(* Logix 5000 project; controller AdvManLab vendor 1 type 14 code 158 rev 28.12; software revision 28.01; part 10 of 13 *)
(* tags used below, declared in another part *)
   R6Z_Assign : BOOL;
   R6Z_Check_InProgress : BOOL;
   R6Z_Check_Part_NO : SINT;
   R6Z_Check_Read : BOOL;
   R6Z_Check_Results : BOOL;
   R6Z_Check_Start : BOOL;
   R6Z_Clear_All : BOOL;
   R6Z_Clear_All_Inprogress : BOOL;
   R6Z_Clear_All_Start : BOOL;
   R6Z_Current_Part_NO : SINT;
   R6Z_Current_Process_NO : SINT;
   R6Z_Part_Type_Counter : SINT;
   R6Z_Process : BOOL;
   R6Z_Read : BOOL;
   R6Z_Read_Check_Fail : BOOL;
   R6Z_Read_Check_InProgress : BOOL;
   R6Z_Read_Check_Results : BOOL;
   R6Z_Read_Check_Start : BOOL;
   R6Z_Read_Finished : BOOL;
   R6Z_Read_InProgress : BOOL;
   R6Z_Read_Results : BOOL;
   R6Z_Read_Start : BOOL;
   R6Z_Write : BOOL;
   R6Z_Write_Finished_Check : BOOL;
   R6Z_Write_Inprogress : BOOL;
   R6Z_Write_Pass : BOOL;
   Cell_2 : Fanuc_Cell;
   CNC_3_Done : BOOL;   // CNC 3 has completed cutting the part
   CNC_4_Done : BOOL;   // CNC 4 has completed cutting the part
   Enable_Process_Update : BOOL;
   Mode_Auto : BOOL;
   Mode_Semi : BOOL;
   Mode_Start : BOOL;
   R2Z_Current_Part_NO : DINT;
   R2Z_Current_Process_NO : DINT;
   R2Z_Read : BOOL;
   R2Z_Read_Finished : BOOL;
   R2Z_Read_InProgress : BOOL;
   R2Z_Read_Results : BOOL;
   R2Z_Read_Start : BOOL;
   R3J_Assign : BOOL;
   R3J_Check_Process_NO : DINT;
   R3J_Current_Part_NO : SINT;
   R3J_Current_Process_NO : SINT;
   R3J_Process : BOOL;
   R3J_Read : BOOL;
   R3J_Read_Check_Fail : BOOL;
   R3J_Read_Check_InProgress : BOOL;
   R3J_Read_Check_Results : BOOL;
   R3J_Read_Check_Start : BOOL;
   R3J_Read_Finished : BOOL;
   R3J_Read_InProgress : BOOL;
   R3J_Read_Results : BOOL;
   R3J_Read_Start : BOOL;
   R3J_Write : BOOL;
   R3J_Write_Finished_Check : BOOL;
   R3J_Write_Inprogress : BOOL;
   R3J_Write_Pass : BOOL;
   R5Z_Current_Part_NO : DINT;
   R5Z_Current_Process_NO : DINT;
   R5Z_Read : BOOL;
   R5Z_Read_Finished : BOOL;
   R5Z_Read_InProgress : BOOL;
   R5Z_Read_Results : BOOL;
   R5Z_Read_Start : BOOL;
   R6S_Check_Current_Part_NO : DINT;
   R6S_Check_Current_Process_NO : DINT;
   R6S_User_Input_Part_NO : DINT;
   R6S_User_Input_Process_NO : DINT;
   R6Z_Check_Read_PB : BOOL;
   R6Z_Clear_All_PB : BOOL;
   R6Z_Write_Check : BOOL;
   R6Z_Write_Check_1 : BOOL;
   R6Z_Write_Inprogress_Check : BOOL;
   R6Z_Write_Inprogress_Check_1 : BOOL;
   R6Z_Write_Test : BOOL;
   R6Z_Write_Test_1 : BOOL;
   R6Z_Write_Test_PB : BOOL;
   RFIDTP2 : ALIAS FOR RFID_N054:I.Channel[1].TagPresent;   // RFID Tag at Cell 2 Hold Back Stop
   RFIDTP3 : ALIAS FOR RFID_N055:I.Channel[0].TagPresent;   // RFID Tag at Cell 2 Stop
   RFIDTP5 : ALIAS FOR RFID_N056:I.Channel[0].TagPresent;   // RFID Tag at Cell 3 Stop
   RFIDTP6 : ALIAS FOR RFID_N056:I.Channel[1].TagPresent;
   Robot2_DroppedP3 : BOOL;
   Robot2_DroppedP4 : BOOL;
   Robot2DroppedPart : BOOL;
(* MainProgram, continued *)

ROUTINE RFID_2_ZZ   (* ladder *)
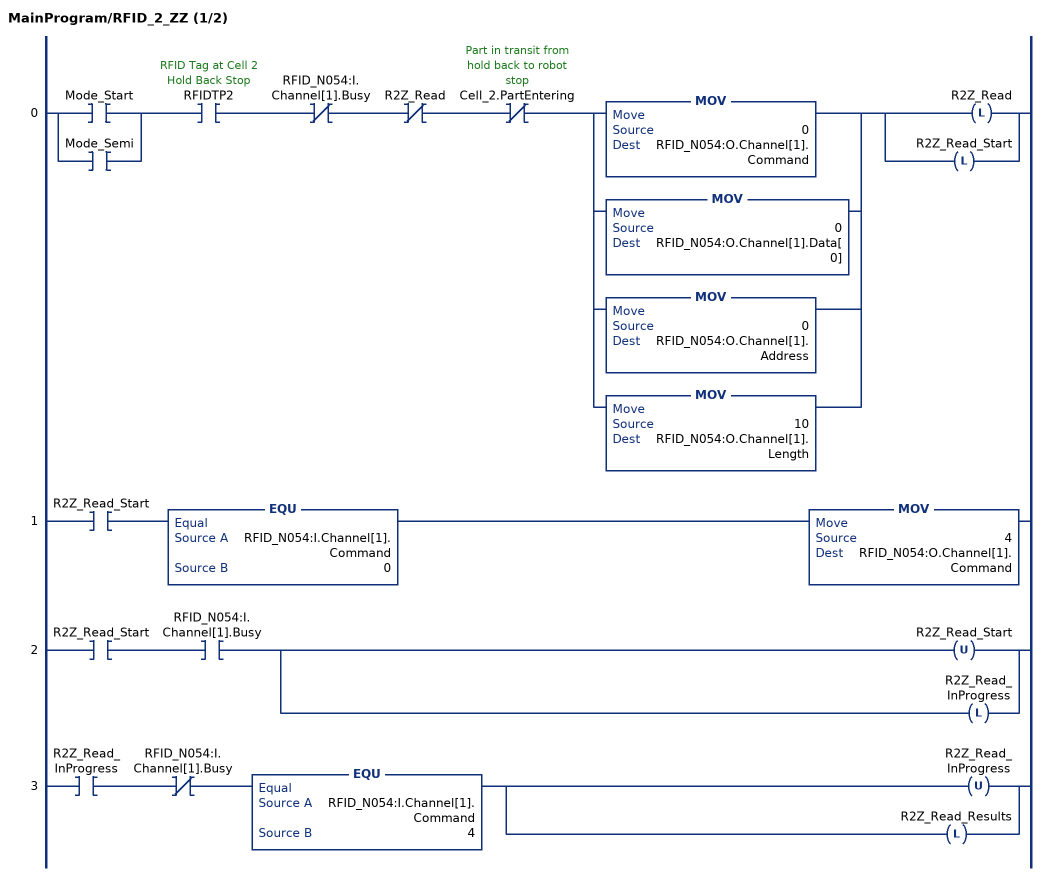
   0: [XIC(Mode_Start) ,XIC(Mode_Semi) ]XIC(RFIDTP2)XIO(RFID_N054:I.Channel[1].Busy)XIO(R2Z_Read)XIO(Cell_2.PartEntering)[MOV(0,RFID_N054:O.Channel[1].Command) ,MOV(0,RFID_N054:O.Channel[1].Data[0]) ,MOV(0,RFID_N054:O.Channel[1].Address) ,MOV(10,RFID_N054:O.Channel[1].Length) ][OTL(R2Z_Read) ,OTL(R2Z_Read_Start) ];
   1: XIC(R2Z_Read_Start)EQU(RFID_N054:I.Channel[1].Command,0)MOV(4,RFID_N054:O.Channel[1].Command);
   2: XIC(R2Z_Read_Start)XIC(RFID_N054:I.Channel[1].Busy)[OTU(R2Z_Read_Start) ,OTL(R2Z_Read_InProgress) ];
   3: XIC(R2Z_Read_InProgress)XIO(RFID_N054:I.Channel[1].Busy)EQU(RFID_N054:I.Channel[1].Command,4)[OTU(R2Z_Read_InProgress) ,OTL(R2Z_Read_Results) ];
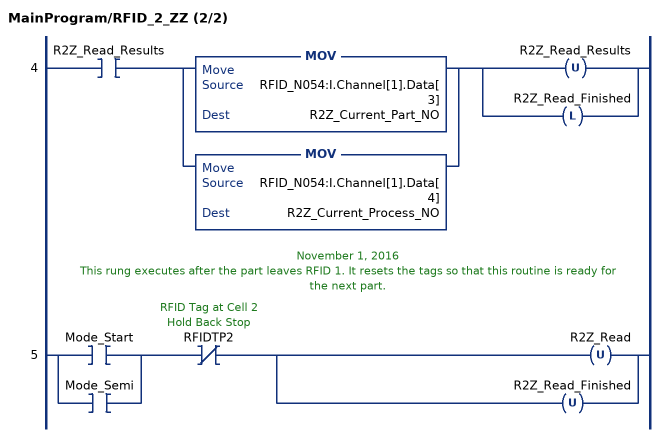
   4: XIC(R2Z_Read_Results)[MOV(RFID_N054:I.Channel[1].Data[3],R2Z_Current_Part_NO) ,MOV(RFID_N054:I.Channel[1].Data[4],R2Z_Current_Process_NO) ][OTU(R2Z_Read_Results) ,OTL(R2Z_Read_Finished) ];
   // November 1, 2016
   // This rung executes after the part leaves RFID 1. It resets the tags so that this routine is ready for the next part.
   5: [XIC(Mode_Start) ,XIC(Mode_Semi) ]XIO(RFIDTP2)[OTU(R2Z_Read) ,OTU(R2Z_Read_Finished) ];
END_ROUTINE

ROUTINE RFID_3_JW   (* ladder *)
// Rewrite of RFID_3 using new read/write logic of RFID_6_ZZ
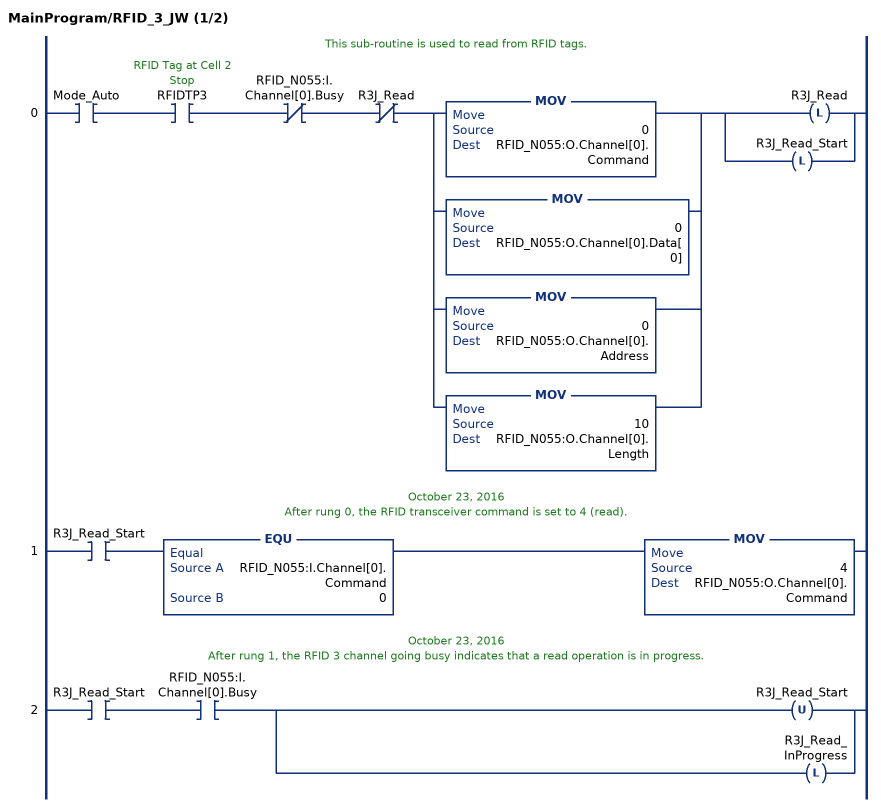
   // This sub-routine is used to read from RFID tags.
   0: XIC(Mode_Auto)XIC(RFIDTP3)XIO(RFID_N055:I.Channel[0].Busy)XIO(R3J_Read)[MOV(0,RFID_N055:O.Channel[0].Command) ,MOV(0,RFID_N055:O.Channel[0].Data[0]) ,MOV(0,RFID_N055:O.Channel[0].Address) ,MOV(10,RFID_N055:O.Channel[0].Length) ][OTL(R3J_Read) ,OTL(R3J_Read_Start) ];
   // October 23, 2016
   // After rung 0, the RFID transceiver command is set to 4 (read).
   1: XIC(R3J_Read_Start)EQU(RFID_N055:I.Channel[0].Command,0)MOV(4,RFID_N055:O.Channel[0].Command);
   // October 23, 2016
   // After rung 1, the RFID 3 channel going busy indicates that a read operation is in progress.
   2: XIC(R3J_Read_Start)XIC(RFID_N055:I.Channel[0].Busy)[OTU(R3J_Read_Start) ,OTL(R3J_Read_InProgress) ];
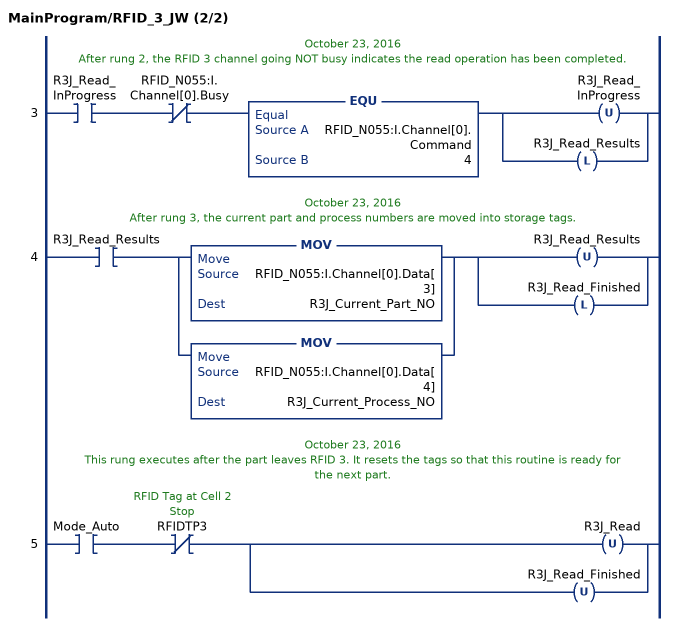
   // October 23, 2016
   // After rung 2, the RFID 3 channel going NOT busy indicates the read operation has been completed.
   3: XIC(R3J_Read_InProgress)XIO(RFID_N055:I.Channel[0].Busy)EQU(RFID_N055:I.Channel[0].Command,4)[OTU(R3J_Read_InProgress) ,OTL(R3J_Read_Results) ];
   // October 23, 2016
   // After rung 3, the current part and process numbers are moved into storage tags.
   4: XIC(R3J_Read_Results)[MOV(RFID_N055:I.Channel[0].Data[3],R3J_Current_Part_NO) ,MOV(RFID_N055:I.Channel[0].Data[4],R3J_Current_Process_NO) ][OTU(R3J_Read_Results) ,OTL(R3J_Read_Finished) ];
   // October 23, 2016
   // This rung executes after the part leaves RFID 3. It resets the tags so that this routine is ready for the next part.
   5: XIC(Mode_Auto)XIO(RFIDTP3)[OTU(R3J_Read) ,OTU(R3J_Read_Finished) ];
END_ROUTINE

ROUTINE RFID_5_ZZ   (* ladder *)
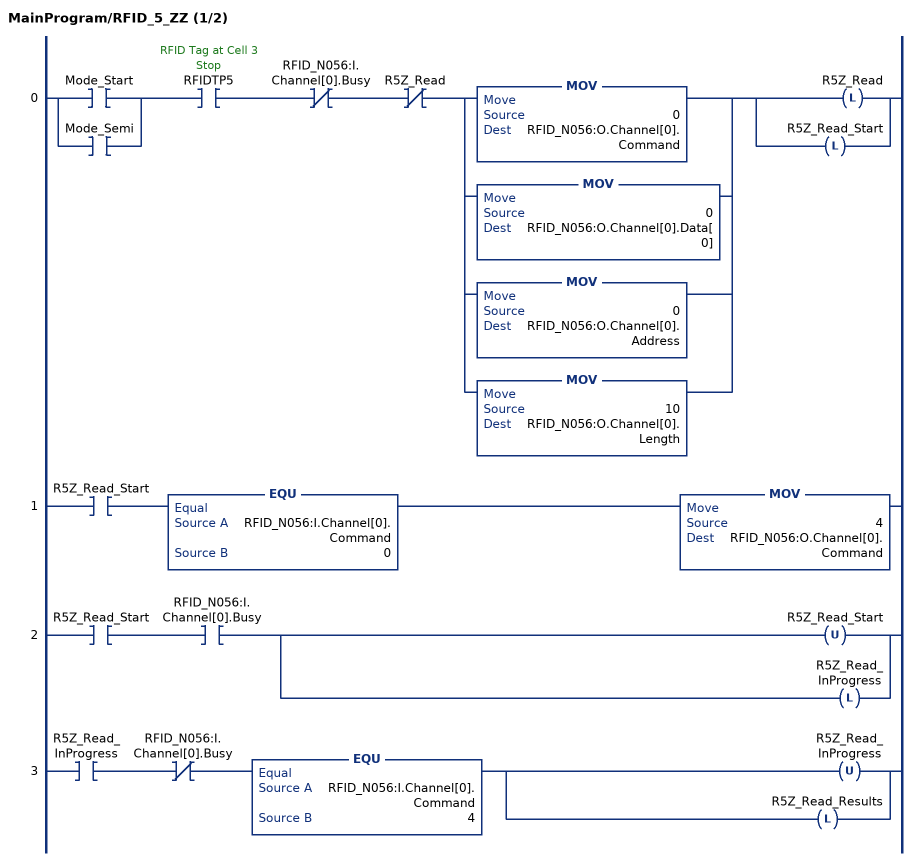
   0: [XIC(Mode_Start) ,XIC(Mode_Semi) ]XIC(RFIDTP5)XIO(RFID_N056:I.Channel[0].Busy)XIO(R5Z_Read)[MOV(0,RFID_N056:O.Channel[0].Command) ,MOV(0,RFID_N056:O.Channel[0].Data[0]) ,MOV(0,RFID_N056:O.Channel[0].Address) ,MOV(10,RFID_N056:O.Channel[0].Length) ][OTL(R5Z_Read) ,OTL(R5Z_Read_Start) ];
   1: XIC(R5Z_Read_Start)EQU(RFID_N056:I.Channel[0].Command,0)MOV(4,RFID_N056:O.Channel[0].Command);
   2: XIC(R5Z_Read_Start)XIC(RFID_N056:I.Channel[0].Busy)[OTU(R5Z_Read_Start) ,OTL(R5Z_Read_InProgress) ];
   3: XIC(R5Z_Read_InProgress)XIO(RFID_N056:I.Channel[0].Busy)EQU(RFID_N056:I.Channel[0].Command,4)[OTU(R5Z_Read_InProgress) ,OTL(R5Z_Read_Results) ];
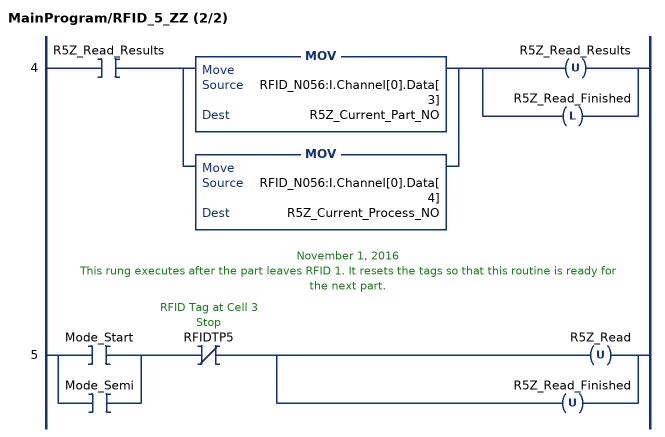
   4: XIC(R5Z_Read_Results)[MOV(RFID_N056:I.Channel[0].Data[3],R5Z_Current_Part_NO) ,MOV(RFID_N056:I.Channel[0].Data[4],R5Z_Current_Process_NO) ][OTU(R5Z_Read_Results) ,OTL(R5Z_Read_Finished) ];
   // November 1, 2016
   // This rung executes after the part leaves RFID 1. It resets the tags so that this routine is ready for the next part.
   5: [XIC(Mode_Start) ,XIC(Mode_Semi) ]XIO(RFIDTP5)[OTU(R5Z_Read) ,OTU(R5Z_Read_Finished) ];
END_ROUTINE

ROUTINE RFID_6_Clear_All_ZZ   (* ladder *)
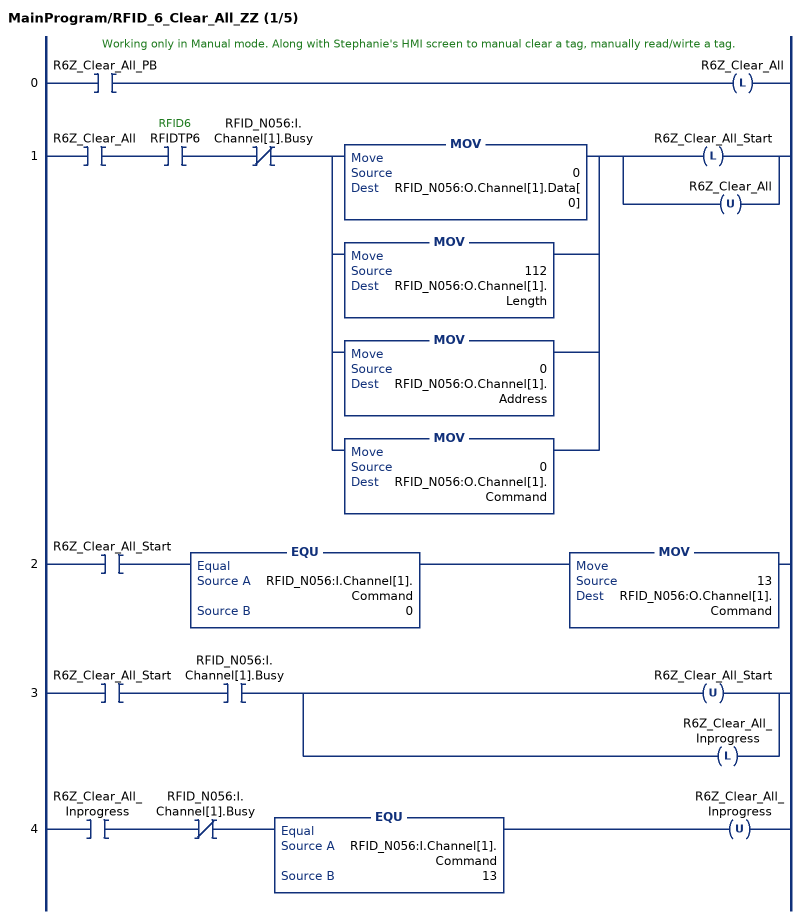
   // Working only in Manual mode. Along with Stephanie's HMI screen to manual clear a tag, manually read/wirte a tag.
   0: XIC(R6Z_Clear_All_PB)OTL(R6Z_Clear_All);
   1: XIC(R6Z_Clear_All)XIC(RFIDTP6)XIO(RFID_N056:I.Channel[1].Busy)[MOV(0,RFID_N056:O.Channel[1].Data[0]) ,MOV(112,RFID_N056:O.Channel[1].Length) ,MOV(0,RFID_N056:O.Channel[1].Address) ,MOV(0,RFID_N056:O.Channel[1].Command) ][OTL(R6Z_Clear_All_Start) ,OTU(R6Z_Clear_All) ];
   2: XIC(R6Z_Clear_All_Start)EQU(RFID_N056:I.Channel[1].Command,0)MOV(13,RFID_N056:O.Channel[1].Command);
   3: XIC(R6Z_Clear_All_Start)XIC(RFID_N056:I.Channel[1].Busy)[OTU(R6Z_Clear_All_Start) ,OTL(R6Z_Clear_All_Inprogress) ];
   4: XIC(R6Z_Clear_All_Inprogress)XIO(RFID_N056:I.Channel[1].Busy)EQU(RFID_N056:I.Channel[1].Command,13)OTU(R6Z_Clear_All_Inprogress);
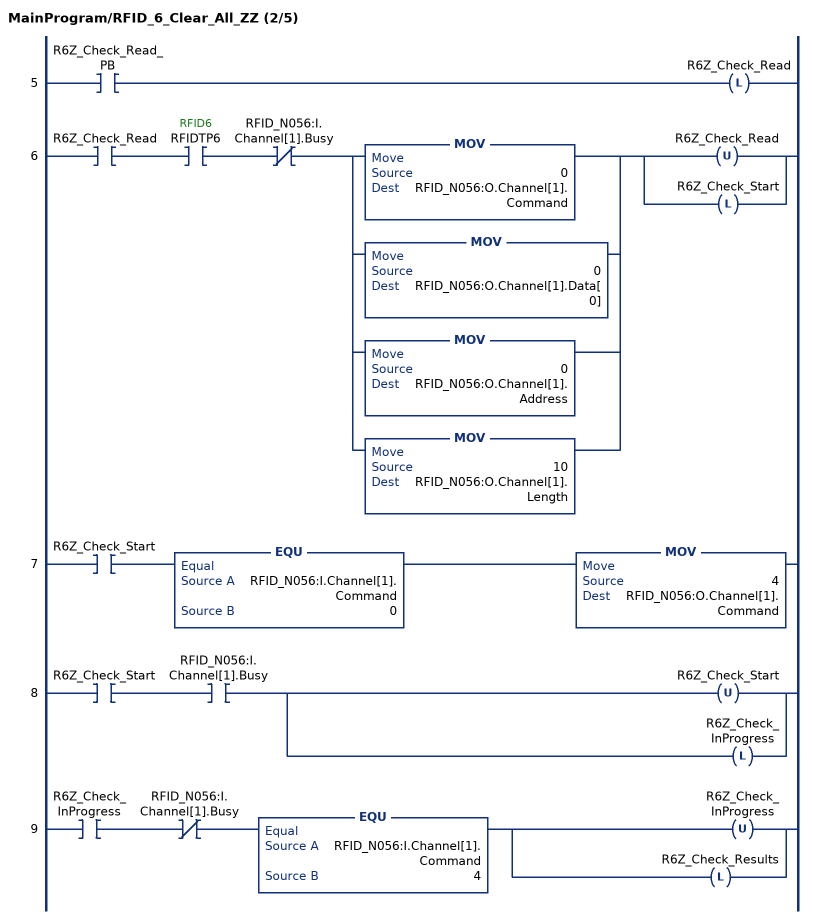
   5: XIC(R6Z_Check_Read_PB)OTL(R6Z_Check_Read);
   6: XIC(R6Z_Check_Read)XIC(RFIDTP6)XIO(RFID_N056:I.Channel[1].Busy)[MOV(0,RFID_N056:O.Channel[1].Command) ,MOV(0,RFID_N056:O.Channel[1].Data[0]) ,MOV(0,RFID_N056:O.Channel[1].Address) ,MOV(10,RFID_N056:O.Channel[1].Length) ][OTU(R6Z_Check_Read) ,OTL(R6Z_Check_Start) ];
   7: XIC(R6Z_Check_Start)EQU(RFID_N056:I.Channel[1].Command,0)MOV(4,RFID_N056:O.Channel[1].Command);
   8: XIC(R6Z_Check_Start)XIC(RFID_N056:I.Channel[1].Busy)[OTU(R6Z_Check_Start) ,OTL(R6Z_Check_InProgress) ];
   9: XIC(R6Z_Check_InProgress)XIO(RFID_N056:I.Channel[1].Busy)EQU(RFID_N056:I.Channel[1].Command,4)[OTU(R6Z_Check_InProgress) ,OTL(R6Z_Check_Results) ];
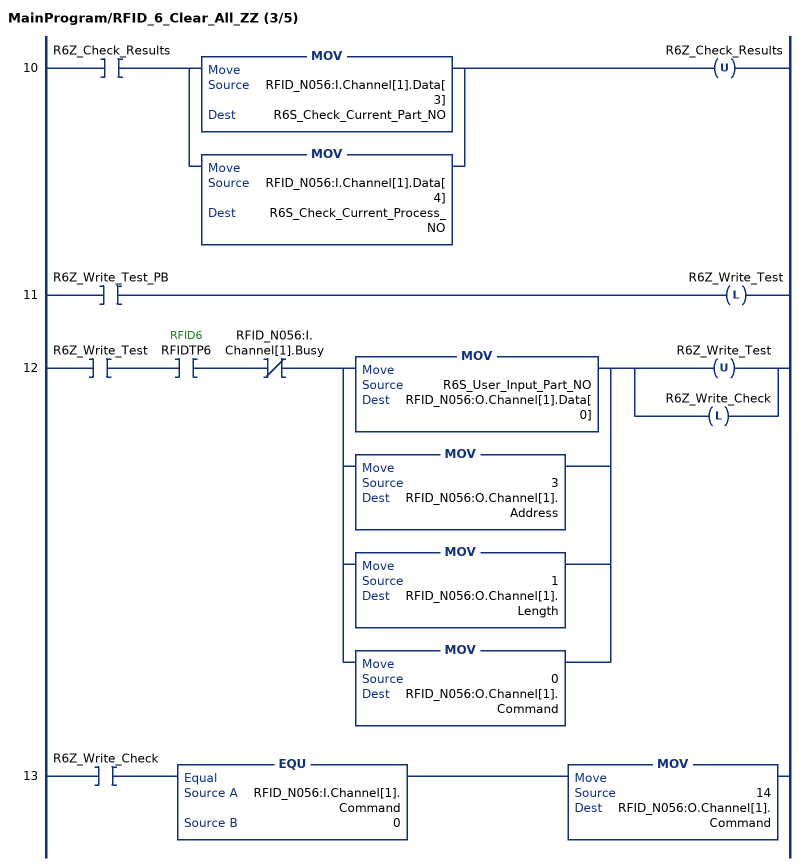
   10: XIC(R6Z_Check_Results)[MOV(RFID_N056:I.Channel[1].Data[3],R6S_Check_Current_Part_NO) ,MOV(RFID_N056:I.Channel[1].Data[4],R6S_Check_Current_Process_NO) ]OTU(R6Z_Check_Results);
   11: XIC(R6Z_Write_Test_PB)OTL(R6Z_Write_Test);
   12: XIC(R6Z_Write_Test)XIC(RFIDTP6)XIO(RFID_N056:I.Channel[1].Busy)[MOV(R6S_User_Input_Part_NO,RFID_N056:O.Channel[1].Data[0]) ,MOV(3,RFID_N056:O.Channel[1].Address) ,MOV(1,RFID_N056:O.Channel[1].Length) ,MOV(0,RFID_N056:O.Channel[1].Command) ][OTU(R6Z_Write_Test) ,OTL(R6Z_Write_Check) ];
   13: XIC(R6Z_Write_Check)EQU(RFID_N056:I.Channel[1].Command,0)MOV(14,RFID_N056:O.Channel[1].Command);
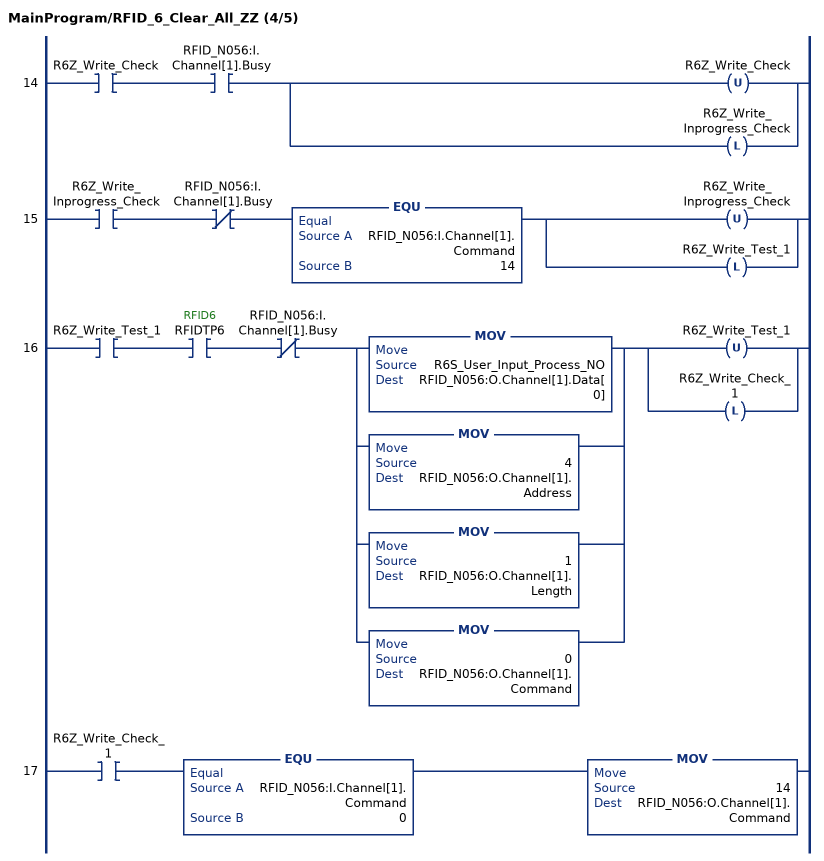
   14: XIC(R6Z_Write_Check)XIC(RFID_N056:I.Channel[1].Busy)[OTU(R6Z_Write_Check) ,OTL(R6Z_Write_Inprogress_Check) ];
   15: XIC(R6Z_Write_Inprogress_Check)XIO(RFID_N056:I.Channel[1].Busy)EQU(RFID_N056:I.Channel[1].Command,14)[OTU(R6Z_Write_Inprogress_Check) ,OTL(R6Z_Write_Test_1) ];
   16: XIC(R6Z_Write_Test_1)XIC(RFIDTP6)XIO(RFID_N056:I.Channel[1].Busy)[MOV(R6S_User_Input_Process_NO,RFID_N056:O.Channel[1].Data[0]) ,MOV(4,RFID_N056:O.Channel[1].Address) ,MOV(1,RFID_N056:O.Channel[1].Length) ,MOV(0,RFID_N056:O.Channel[1].Command) ][OTU(R6Z_Write_Test_1) ,OTL(R6Z_Write_Check_1) ];
   17: XIC(R6Z_Write_Check_1)EQU(RFID_N056:I.Channel[1].Command,0)MOV(14,RFID_N056:O.Channel[1].Command);
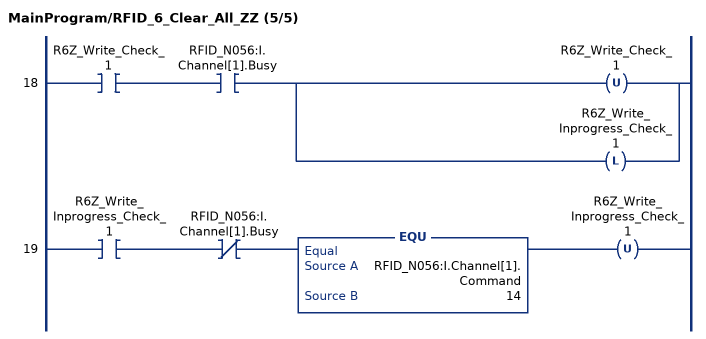
   18: XIC(R6Z_Write_Check_1)XIC(RFID_N056:I.Channel[1].Busy)[OTU(R6Z_Write_Check_1) ,OTL(R6Z_Write_Inprogress_Check_1) ];
   19: XIC(R6Z_Write_Inprogress_Check_1)XIO(RFID_N056:I.Channel[1].Busy)EQU(RFID_N056:I.Channel[1].Command,14)OTU(R6Z_Write_Inprogress_Check_1);
END_ROUTINE

ROUTINE RFID_6_ZZ   (* ladder *)
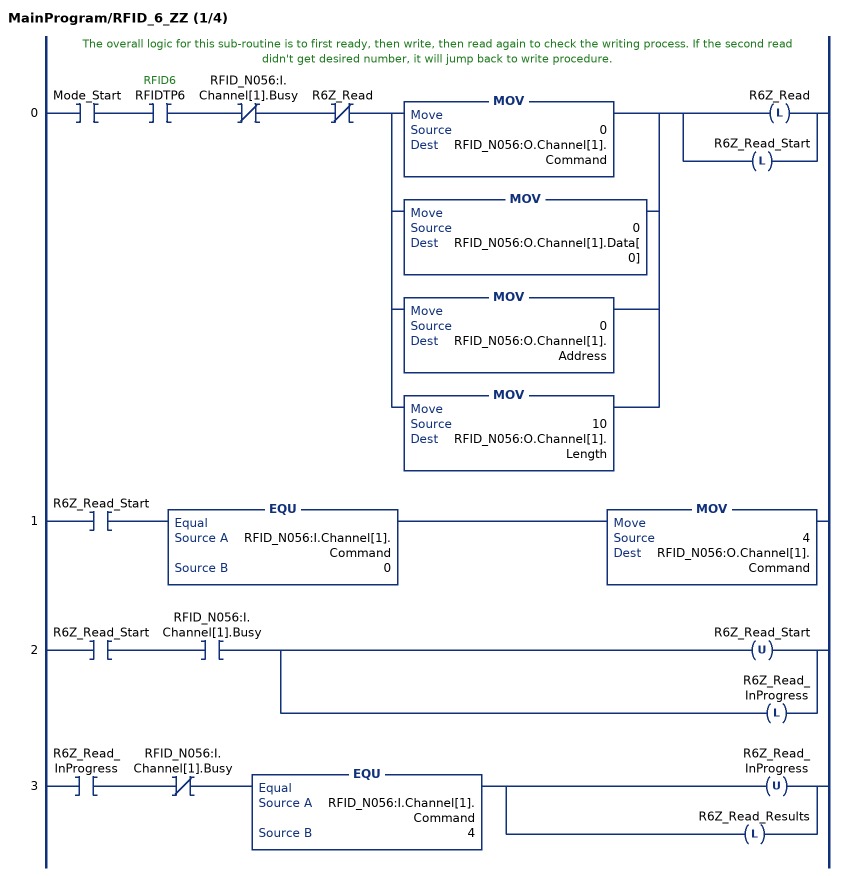
   // The overall logic for this sub-routine is to first ready, then write, then read again to check the writing process. If the second read didn't get desired number, it will jump back to write procedure.
   0: XIC(Mode_Start)XIC(RFIDTP6)XIO(RFID_N056:I.Channel[1].Busy)XIO(R6Z_Read)[MOV(0,RFID_N056:O.Channel[1].Command) ,MOV(0,RFID_N056:O.Channel[1].Data[0]) ,MOV(0,RFID_N056:O.Channel[1].Address) ,MOV(10,RFID_N056:O.Channel[1].Length) ][OTL(R6Z_Read) ,OTL(R6Z_Read_Start) ];
   1: XIC(R6Z_Read_Start)EQU(RFID_N056:I.Channel[1].Command,0)MOV(4,RFID_N056:O.Channel[1].Command);
   2: XIC(R6Z_Read_Start)XIC(RFID_N056:I.Channel[1].Busy)[OTU(R6Z_Read_Start) ,OTL(R6Z_Read_InProgress) ];
   3: XIC(R6Z_Read_InProgress)XIO(RFID_N056:I.Channel[1].Busy)EQU(RFID_N056:I.Channel[1].Command,4)[OTU(R6Z_Read_InProgress) ,OTL(R6Z_Read_Results) ];
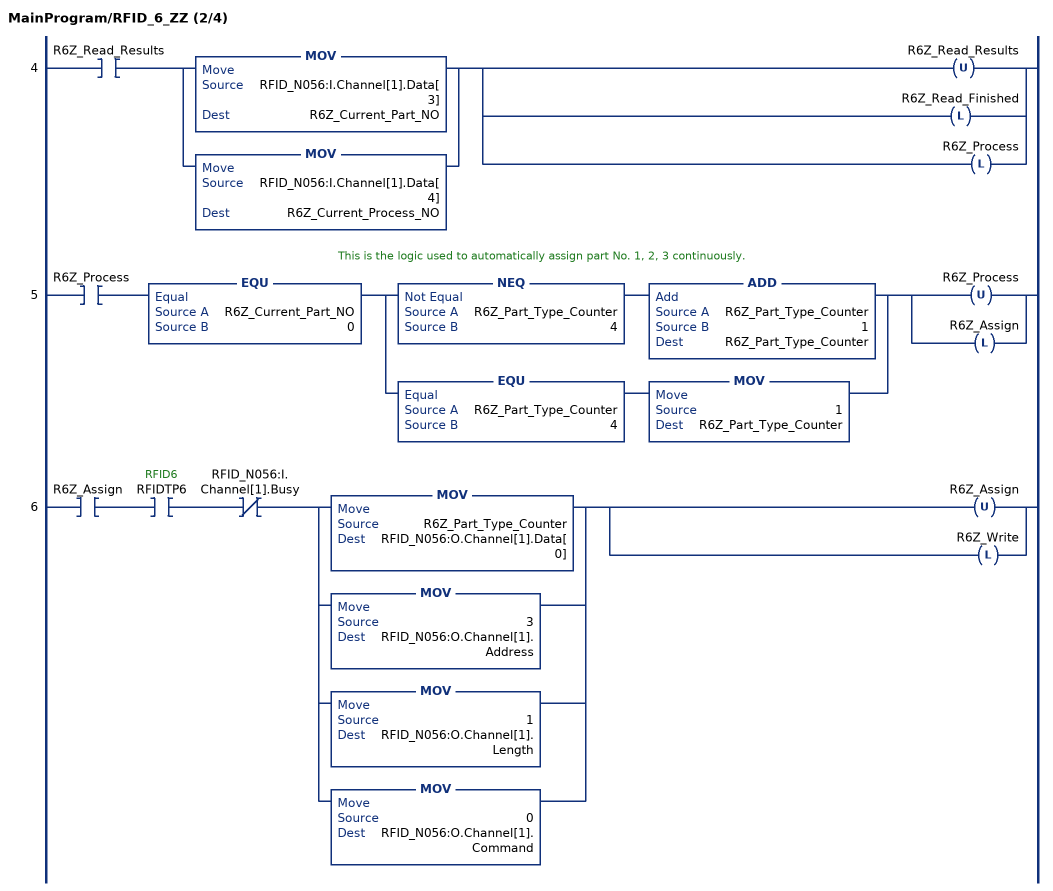
   4: XIC(R6Z_Read_Results)[MOV(RFID_N056:I.Channel[1].Data[3],R6Z_Current_Part_NO) ,MOV(RFID_N056:I.Channel[1].Data[4],R6Z_Current_Process_NO) ][OTU(R6Z_Read_Results) ,OTL(R6Z_Read_Finished) ,OTL(R6Z_Process) ];
   // This is the logic used to automatically assign part No. 1, 2, 3 continuously.
   5: XIC(R6Z_Process)EQU(R6Z_Current_Part_NO,0)[NEQ(R6Z_Part_Type_Counter,4) ADD(R6Z_Part_Type_Counter,1,R6Z_Part_Type_Counter) ,EQU(R6Z_Part_Type_Counter,4) MOV(1,R6Z_Part_Type_Counter) ][OTU(R6Z_Process) ,OTL(R6Z_Assign) ];
   6: XIC(R6Z_Assign)XIC(RFIDTP6)XIO(RFID_N056:I.Channel[1].Busy)[MOV(R6Z_Part_Type_Counter,RFID_N056:O.Channel[1].Data[0]) ,MOV(3,RFID_N056:O.Channel[1].Address) ,MOV(1,RFID_N056:O.Channel[1].Length) ,MOV(0,RFID_N056:O.Channel[1].Command) ][OTU(R6Z_Assign) ,OTL(R6Z_Write) ];
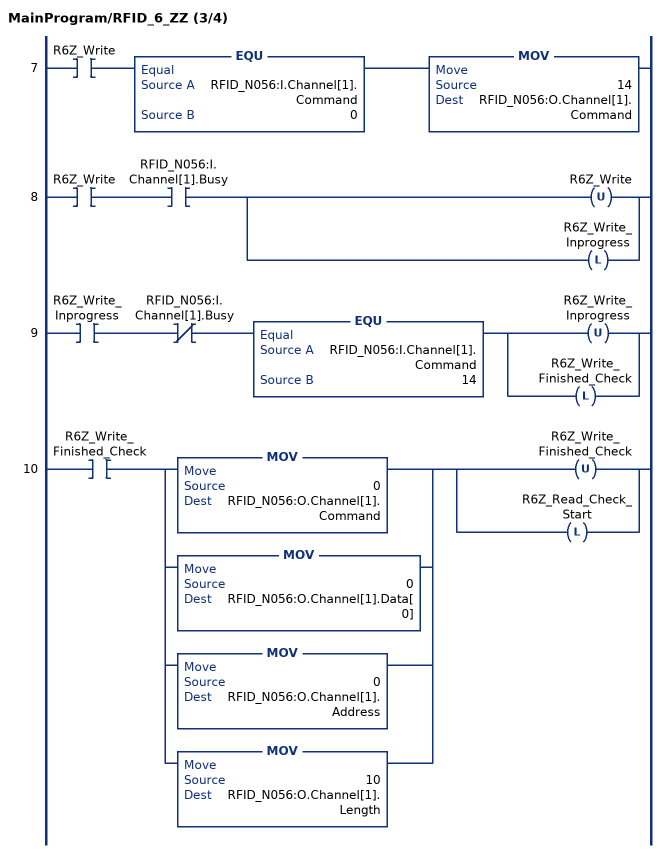
   7: XIC(R6Z_Write)EQU(RFID_N056:I.Channel[1].Command,0)MOV(14,RFID_N056:O.Channel[1].Command);
   8: XIC(R6Z_Write)XIC(RFID_N056:I.Channel[1].Busy)[OTU(R6Z_Write) ,OTL(R6Z_Write_Inprogress) ];
   9: XIC(R6Z_Write_Inprogress)XIO(RFID_N056:I.Channel[1].Busy)EQU(RFID_N056:I.Channel[1].Command,14)[OTU(R6Z_Write_Inprogress) ,OTL(R6Z_Write_Finished_Check) ];
   10: XIC(R6Z_Write_Finished_Check)[MOV(0,RFID_N056:O.Channel[1].Command) ,MOV(0,RFID_N056:O.Channel[1].Data[0]) ,MOV(0,RFID_N056:O.Channel[1].Address) ,MOV(10,RFID_N056:O.Channel[1].Length) ][OTU(R6Z_Write_Finished_Check) ,OTL(R6Z_Read_Check_Start) ];
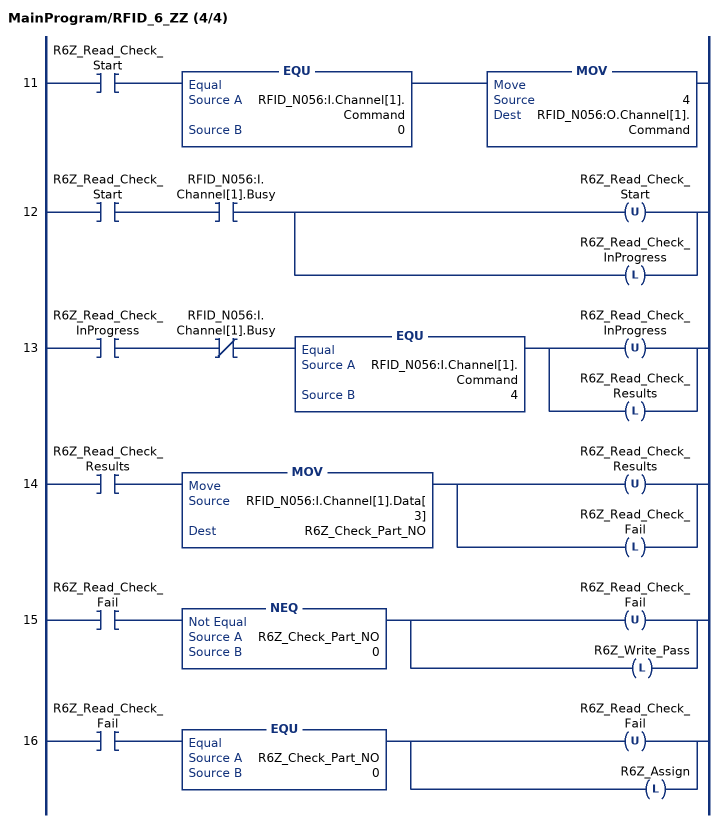
   11: XIC(R6Z_Read_Check_Start)EQU(RFID_N056:I.Channel[1].Command,0)MOV(4,RFID_N056:O.Channel[1].Command);
   12: XIC(R6Z_Read_Check_Start)XIC(RFID_N056:I.Channel[1].Busy)[OTU(R6Z_Read_Check_Start) ,OTL(R6Z_Read_Check_InProgress) ];
   13: XIC(R6Z_Read_Check_InProgress)XIO(RFID_N056:I.Channel[1].Busy)EQU(RFID_N056:I.Channel[1].Command,4)[OTU(R6Z_Read_Check_InProgress) ,OTL(R6Z_Read_Check_Results) ];
   14: XIC(R6Z_Read_Check_Results)MOV(RFID_N056:I.Channel[1].Data[3],R6Z_Check_Part_NO)[OTU(R6Z_Read_Check_Results) ,OTL(R6Z_Read_Check_Fail) ];
   15: XIC(R6Z_Read_Check_Fail)NEQ(R6Z_Check_Part_NO,0)[OTU(R6Z_Read_Check_Fail) ,OTL(R6Z_Write_Pass) ];
   16: XIC(R6Z_Read_Check_Fail)EQU(R6Z_Check_Part_NO,0)[OTU(R6Z_Read_Check_Fail) ,OTL(R6Z_Assign) ];
END_ROUTINE

ROUTINE RFID_BU   (* ladder *)
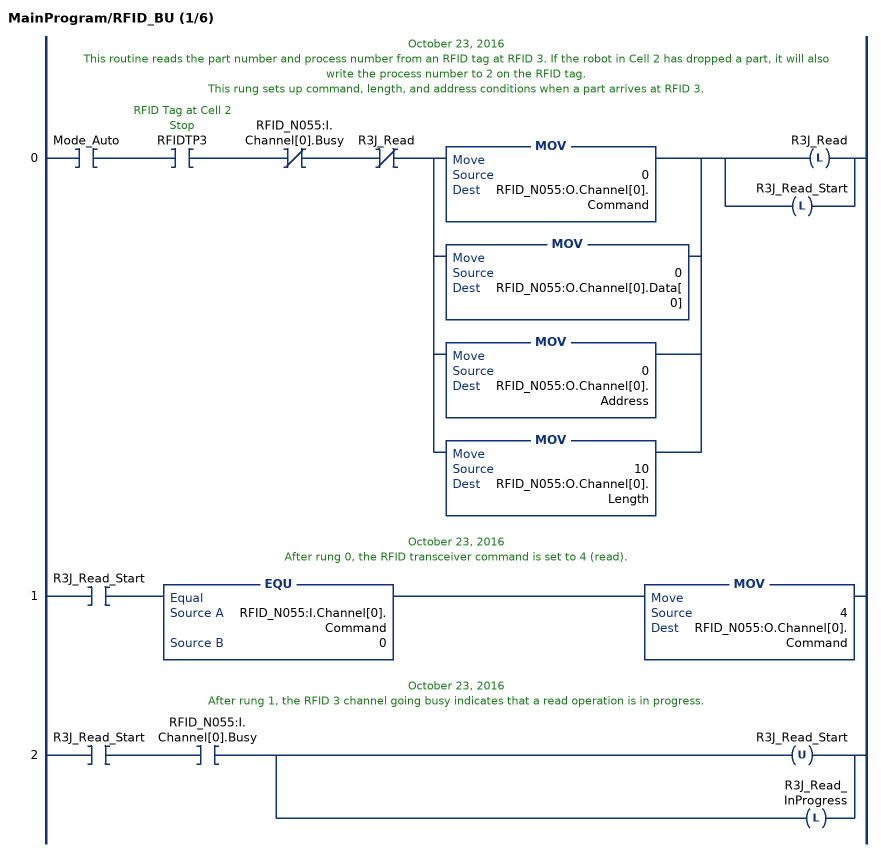
   // October 23, 2016
   // This routine reads the part number and process number from an RFID tag at RFID 3. If the robot in Cell 2 has dropped a part, it will also write the process number to 2 on the RFID tag.
   // This rung sets up command, length, and address conditions when a part arrives at RFID 3.
   0: XIC(Mode_Auto)XIC(RFIDTP3)XIO(RFID_N055:I.Channel[0].Busy)XIO(R3J_Read)[MOV(0,RFID_N055:O.Channel[0].Command) ,MOV(0,RFID_N055:O.Channel[0].Data[0]) ,MOV(0,RFID_N055:O.Channel[0].Address) ,MOV(10,RFID_N055:O.Channel[0].Length) ][OTL(R3J_Read) ,OTL(R3J_Read_Start) ];
   // October 23, 2016
   // After rung 0, the RFID transceiver command is set to 4 (read).
   1: XIC(R3J_Read_Start)EQU(RFID_N055:I.Channel[0].Command,0)MOV(4,RFID_N055:O.Channel[0].Command);
   // October 23, 2016
   // After rung 1, the RFID 3 channel going busy indicates that a read operation is in progress.
   2: XIC(R3J_Read_Start)XIC(RFID_N055:I.Channel[0].Busy)[OTU(R3J_Read_Start) ,OTL(R3J_Read_InProgress) ];
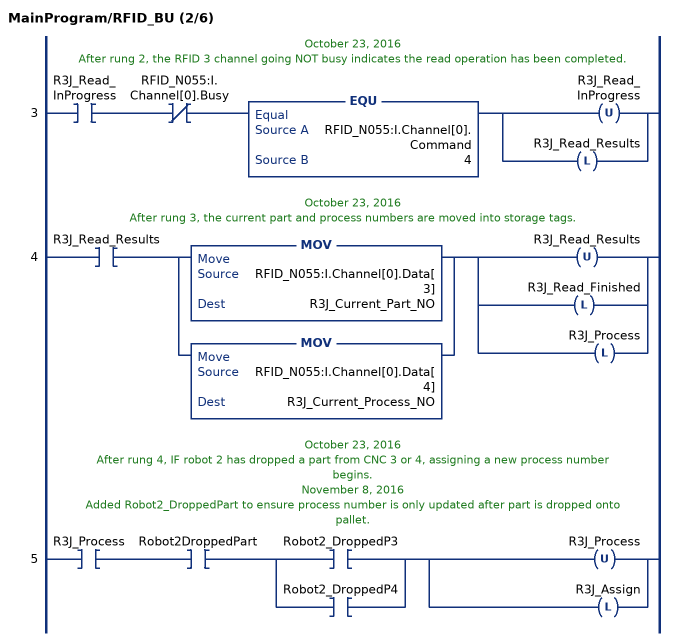
   // October 23, 2016
   // After rung 2, the RFID 3 channel going NOT busy indicates the read operation has been completed.
   3: XIC(R3J_Read_InProgress)XIO(RFID_N055:I.Channel[0].Busy)EQU(RFID_N055:I.Channel[0].Command,4)[OTU(R3J_Read_InProgress) ,OTL(R3J_Read_Results) ];
   // October 23, 2016
   // After rung 3, the current part and process numbers are moved into storage tags.
   4: XIC(R3J_Read_Results)[MOV(RFID_N055:I.Channel[0].Data[3],R3J_Current_Part_NO) ,MOV(RFID_N055:I.Channel[0].Data[4],R3J_Current_Process_NO) ][OTU(R3J_Read_Results) ,OTL(R3J_Read_Finished) ,OTL(R3J_Process) ];
   // October 23, 2016
   // After rung 4, IF robot 2 has dropped a part from CNC 3 or 4, assigning a new process number begins.
   // November 8, 2016
   // Added Robot2_DroppedPart to ensure process number is only updated after part is dropped onto pallet.
   5: XIC(R3J_Process)XIC(Robot2DroppedPart)[XIC(Robot2_DroppedP3) ,XIC(Robot2_DroppedP4) ][OTU(R3J_Process) ,OTL(R3J_Assign) ];
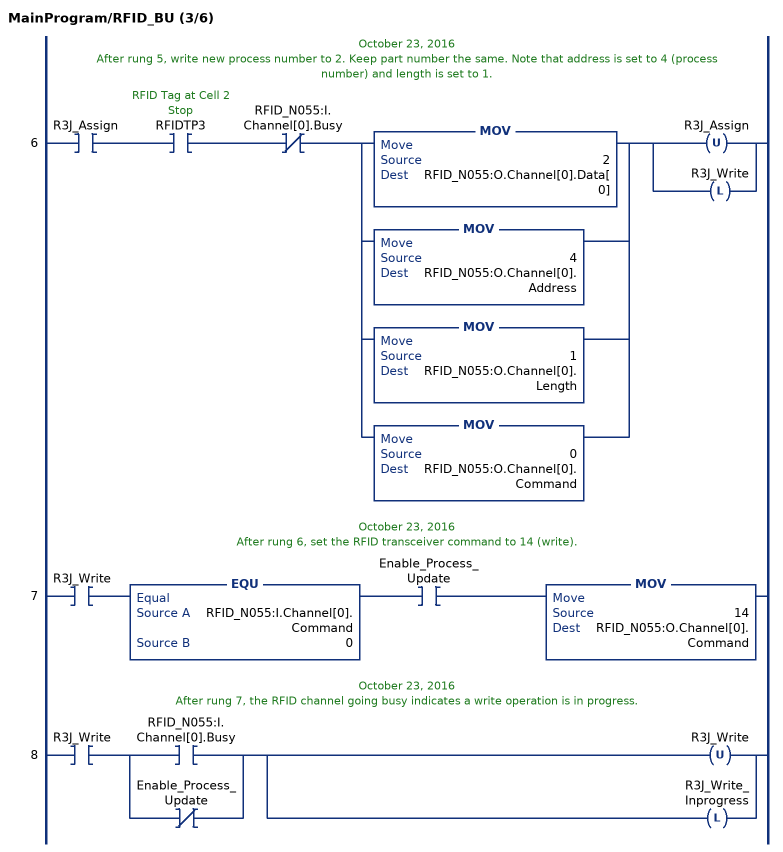
   // October 23, 2016
   // After rung 5, write new process number to 2. Keep part number the same. Note that address is set to 4 (process number) and length is set to 1.
   6: XIC(R3J_Assign)XIC(RFIDTP3)XIO(RFID_N055:I.Channel[0].Busy)[MOV(2,RFID_N055:O.Channel[0].Data[0]) ,MOV(4,RFID_N055:O.Channel[0].Address) ,MOV(1,RFID_N055:O.Channel[0].Length) ,MOV(0,RFID_N055:O.Channel[0].Command) ][OTU(R3J_Assign) ,OTL(R3J_Write) ];
   // October 23, 2016
   // After rung 6, set the RFID transceiver command to 14 (write).
   7: XIC(R3J_Write)EQU(RFID_N055:I.Channel[0].Command,0)XIC(Enable_Process_Update)MOV(14,RFID_N055:O.Channel[0].Command);
   // October 23, 2016
   // After rung 7, the RFID channel going busy indicates a write operation is in progress.
   8: XIC(R3J_Write)[XIC(RFID_N055:I.Channel[0].Busy) ,XIO(Enable_Process_Update) ][OTU(R3J_Write) ,OTL(R3J_Write_Inprogress) ];
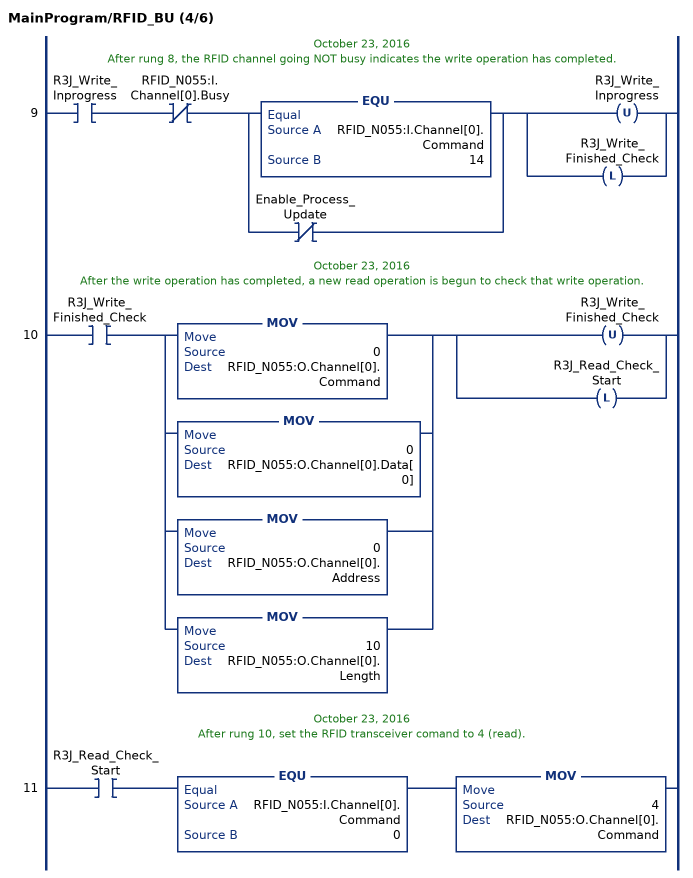
   // October 23, 2016
   // After rung 8, the RFID channel going NOT busy indicates the write operation has completed.
   9: XIC(R3J_Write_Inprogress)XIO(RFID_N055:I.Channel[0].Busy)[EQU(RFID_N055:I.Channel[0].Command,14) ,XIO(Enable_Process_Update) ][OTU(R3J_Write_Inprogress) ,OTL(R3J_Write_Finished_Check) ];
   // October 23, 2016
   // After the write operation has completed, a new read operation is begun to check that write operation.
   10: XIC(R3J_Write_Finished_Check)[MOV(0,RFID_N055:O.Channel[0].Command) ,MOV(0,RFID_N055:O.Channel[0].Data[0]) ,MOV(0,RFID_N055:O.Channel[0].Address) ,MOV(10,RFID_N055:O.Channel[0].Length) ][OTU(R3J_Write_Finished_Check) ,OTL(R3J_Read_Check_Start) ];
   // October 23, 2016
   // After rung 10, set the RFID transceiver comand to 4 (read).
   11: XIC(R3J_Read_Check_Start)EQU(RFID_N055:I.Channel[0].Command,0)MOV(4,RFID_N055:O.Channel[0].Command);
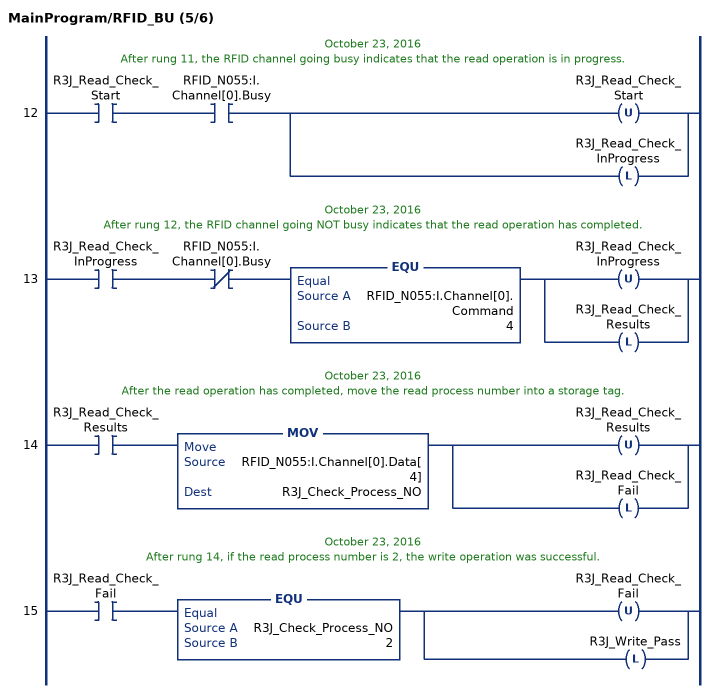
   // October 23, 2016
   // After rung 11, the RFID channel going busy indicates that the read operation is in progress.
   12: XIC(R3J_Read_Check_Start)XIC(RFID_N055:I.Channel[0].Busy)[OTU(R3J_Read_Check_Start) ,OTL(R3J_Read_Check_InProgress) ];
   // October 23, 2016
   // After rung 12, the RFID channel going NOT busy indicates that the read operation has completed.
   13: XIC(R3J_Read_Check_InProgress)XIO(RFID_N055:I.Channel[0].Busy)EQU(RFID_N055:I.Channel[0].Command,4)[OTU(R3J_Read_Check_InProgress) ,OTL(R3J_Read_Check_Results) ];
   // October 23, 2016
   // After the read operation has completed, move the read process number into a storage tag.
   14: XIC(R3J_Read_Check_Results)MOV(RFID_N055:I.Channel[0].Data[4],R3J_Check_Process_NO)[OTU(R3J_Read_Check_Results) ,OTL(R3J_Read_Check_Fail) ];
   // October 23, 2016
   // After rung 14, if the read process number is 2, the write operation was successful.
   15: XIC(R3J_Read_Check_Fail)EQU(R3J_Check_Process_NO,2)[OTU(R3J_Read_Check_Fail) ,OTL(R3J_Write_Pass) ];
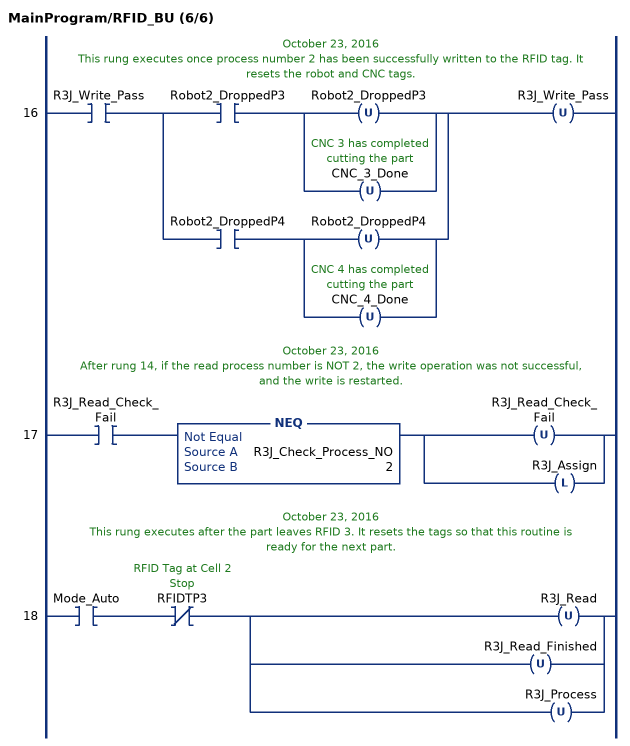
   // October 23, 2016
   // This rung executes once process number 2 has been successfully written to the RFID tag. It resets the robot and CNC tags.
   16: XIC(R3J_Write_Pass)[XIC(Robot2_DroppedP3) [OTU(Robot2_DroppedP3) ,OTU(CNC_3_Done) ] ,XIC(Robot2_DroppedP4) [OTU(Robot2_DroppedP4) ,OTU(CNC_4_Done) ] ]OTU(R3J_Write_Pass);
   // October 23, 2016
   // After rung 14, if the read process number is NOT 2, the write operation was not successful, and the write is restarted.
   17: XIC(R3J_Read_Check_Fail)NEQ(R3J_Check_Process_NO,2)[OTU(R3J_Read_Check_Fail) ,OTL(R3J_Assign) ];
   // October 23, 2016
   // This rung executes after the part leaves RFID 3. It resets the tags so that this routine is ready for the next part.
   18: XIC(Mode_Auto)XIO(RFIDTP3)[OTU(R3J_Read) ,OTU(R3J_Read_Finished) ,OTU(R3J_Process) ];
END_ROUTINE
